Fanuc KAREL source: kd00069.KL

-- PROVISIONAL review KL for V1013-1; original PC SHA256 46b11d614ca88db647ee1a5f5f84015ac4c7d4ff12067eec14543316ff3cc67f
-- Incomplete behavior may be omitted. Consult companion uncertainty JSON. Do not deploy.
PROGRAM KD00069
%NOLOCKGROUP
VAR
  I : INTEGER
  J : INTEGER
  B : BOOLEAN
  R : REAL
  S : STRING[80]
BEGIN
  -- UNRESOLVED_PC offsets 5-18; opcodes 9D,81,18,9D,1B,9D,12,9C,13,04
  -- UNRESOLVED_PC offsets 23-27; opcodes 7F
END KD00069
